// TIA Portal V18 export
// export: Created 2025-12-01T17:53:13.1665706Z, ExportSetting None, DisplayName Totally Integrated Automation Portal, DisplayVersion V18 Update 5, DisplayName TIA Portal Openness, DisplayVersion V18 Update 5, DisplayName TIA Portal Teamcenter Gateway, DisplayVersion V18, DisplayName TIA Portal Version Control Interface, DisplayVersion V18, DisplayName STEP 7 Professional, DisplayVersion V18 Update 5, DisplayName STEP 7 Safety, DisplayVersion V18, DisplayName WinCC Professional, DisplayVersion V18 Update 5
Screen "800Main"  1280x800, Number=800, Template=08CtrlPanel
  ScreenLayer "Layer_0"
    Button "按钮_9"  PictureOff=向右箭头_0, StyleItem=BtnFunction20, TextOff="停止 运行系统 / Stop Runtime / Zastaviť Runtime", TextOn="停止 运行系统 / Stop Runtime / Zastaviť Runtime"
      on Click: StopRuntime(Mode := 0)
    Button "按钮_5"  PictureOff=向右箭头_0, StyleItem=BtnFunction20, TextOff="打开控 制面板 / GoToControl Panel / Prejsť na ovládanie Panel"
      on Click: OpenControlPanel()
    Button "按钮_10"  PictureOff=向右箭头_0, StyleItem=BtnFunction20, TextOff="清屏 / Clear Panel / Jasný Panel", TextOn="清屏 / Clear Panel / Jasný Panel"
      on Release: ActivateCleanScreen(Time period := 30)
    Switch "开关_1" at 1152,95 size 128x75  Mode=TextSwitchButton, StyleItem=Switch20, CaptionText="Switch / Prepínač", TextOff="蜂鸣器 打开 / Buzzer ON / Bzučiak NA", TextOn="蜂鸣器 关闭 / Buzzer OFF / Bzučiak PREČ"
      RangeAppearanceAnimation "RangeAppearanceAnimation"
        tag ST_CommandBuzzerOn
        1..1: back #8bafd3, fore #000000, flashing
      ProcessValue := ST_CommandBuzzerOn
    Button "按钮_1" at 128,725 size 128x75  Authorization=System config, StyleItem=BtnActive20, TextOff="控制面板 / Control Panel / Ovládať Panel"
      on Click: ActivateScreen(Screen name := , Object number := 0); SetTag(Tag := Sys_VersionManagement_HMIPageID, Value := 800)
    Button "按钮_2"  StyleItem=BtnFunction20, TextOff="校准 / Caliration / Kalibrácia"
      on Click: CalibrateTouchScreen()
    Button "btnMenu8_2"  StyleItem=BtnFunction20
    Button "按钮_3"  StyleItem=BtnFunction20, TextOff="显示软件 版本 / Veision Indicator / Veision Indikátor"
      on Click: ShowSoftwareVersion(Display mode := -1)
    Button "按钮_4" at 1152,180 size 128x75  StyleItem=BtnFunction20
    Button "btnMenu8_1" at 1152,350 size 128x75  StyleItem=BtnFunction20, TextOff="配方备份 / Recipe backup / Zálohovanie receptov"
      on Click: ExportDataRecords(Recipe number/name := 1, Data record number/name := 0, File name := \Storage Card USB\record.csv, Overwrite := 2, Output status message := 1, Processing status := )
    Button "按钮_6" at 1152,265 size 128x75  StyleItem=BtnFunction20
    Button "btnMenu8_3" at 1152,520 size 128x75  StyleItem=BtnFunction20
    Button "按钮_7" at 1152,435 size 128x75  StyleItem=BtnFunction20, TextOff="配方恢复 / Recipe recovery / Obnova receptu"
      on Click: ImportDataRecords(File name := \Storage Card USB\record.csv, Data record number/name := 0, Overwrite := 2, Output status message := 1, Processing status := )
    Button "btnMenu8_5"  StyleItem=BtnFunction20
    Button "btnMenu8_6" at 1152,605 size 128x75  StyleItem=BtnFunction20
  ScreenLayer 
  ScreenLayer 
  ScreenLayer 
  ScreenLayer 
  ScreenLayer 
  ScreenLayer 
  ScreenLayer 
  ScreenLayer 
  ScreenLayer 
  ScreenLayer 
  ScreenLayer 
  ScreenLayer 
  ScreenLayer 
  ScreenLayer 
  ScreenLayer 
  ScreenLayer 
  ScreenLayer 
  ScreenLayer 
  ScreenLayer 
  ScreenLayer 
  ScreenLayer 
  ScreenLayer 
  ScreenLayer 
  ScreenLayer 
  ScreenLayer 
  ScreenLayer 
  ScreenLayer 
  ScreenLayer 
  ScreenLayer 
  ScreenLayer 
  ScreenLayer 
